INTERFACE I_Pump

END_INTERFACE

(* stored: Version 1.1.0.1, ProductVersion 3.1.4024.16
   Itf I_Pump: Id {ad974786-fce1-44bd-840c-12d16c9b66d4} *)
